{attribute 'GeneratedUsingTerminal: CX5010 EtherCAT slave-1b82-0016'}
{attribute addProperty BoxType "CX5010 EtherCAT slave-1b82-0016"}
{attribute addProperty Id "TxPdoStateAT %I*BOOL1TxPdoToggleAT %I*BOOL1"}
{attribute addProperty CRC "1643614327"}
{attribute addProperty Size "2"}
TYPE Device_Status_Mapping_61F79077 :
STRUCT
	{attribute addProperty Name "TxPdoState"}
	TxPdoState AT %I* : BOOL;
	{attribute addProperty Name "TxPdoToggle"}
	TxPdoToggle AT %I* : BOOL;
END_STRUCT
END_TYPE

(* stored: Version 1.2.0.0, ProductVersion 3.1.4024.9
   DUT Device_Status_Mapping_61F79077: Id {8de3f18b-fb25-4c44-b01e-a15306965833} *)
